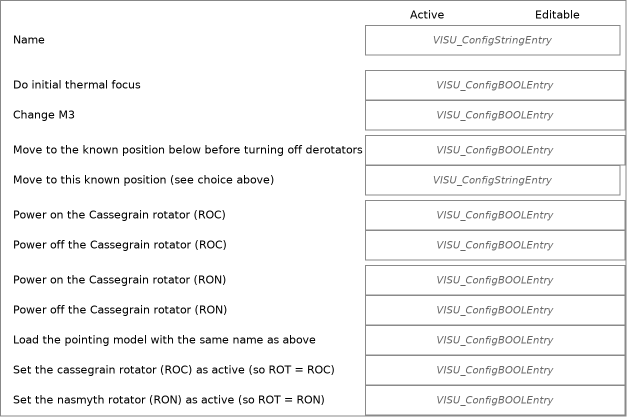
VISUALIZATION VISU_MTCSConfig_Instrument  // 627x417
VAR_IN_OUT
    active : InstrumentConfig;
    editable : InstrumentConfig;
END_VAR
    Label (365,5 125x20), "Active"
    Label (495,5 125x20), "Editable"
    Label (10,25 125x30), "Name"
    Frame (365,25 255x30)
        shows VISU_ConfigStringEntry(active := active.name, editable := editable.name)
    Label (10,70 160x30), "Do initial thermal focus"
    Frame (365,70 260x30)
        shows VISU_ConfigBOOLEntry(active := active.doInitialThermalFocus, editable := editable.doInitialThermalFocus)
    Label (10,100 160x30), "Change M3"
    Frame (365,100 260x30)
        shows VISU_ConfigBOOLEntry(active := active.changeM3, editable := editable.changeM3)
    Frame (365,135 260x30)
        shows VISU_ConfigBOOLEntry(active := active.moveKnownPosition, editable := editable.moveKnownPosition)
    Label (10,135 360x30), "Move to the known position below before turning off derotators"
    Frame (365,200 260x30)
        shows VISU_ConfigBOOLEntry(active := active.powerOnRoc, editable := editable.powerOnRoc)
    Label (10,200 280x30), "Power on the Cassegrain rotator (ROC)"
    Frame (365,165 255x30)
        shows VISU_ConfigStringEntry(active := active.moveKnownPositionName, editable := editable.moveKnownPositionName)
    Label (10,165 340x30), "Move to this known position (see choice above)"
    Frame (365,230 260x30)
        shows VISU_ConfigBOOLEntry(active := active.powerOffRoc, editable := editable.powerOffRoc)
    Label (10,230 350x30), "Power off the Cassegrain rotator (ROC)"
    Frame (365,265 260x30)
        shows VISU_ConfigBOOLEntry(active := active.powerOnRon, editable := editable.powerOnRon)
    Label (10,265 280x30), "Power on the Cassegrain rotator (RON)"
    Frame (365,295 260x30)
        shows VISU_ConfigBOOLEntry(active := active.powerOffRon, editable := editable.powerOffRon)
    Label (10,295 350x30), "Power off the Cassegrain rotator (RON)"
    Frame (365,325 260x30)
        shows VISU_ConfigBOOLEntry(active := active.loadPointingModel, editable := editable.loadPointingModel)
    Label (10,325 360x30), "Load the pointing model with the same name as above"
    Label (10,355 360x30), "Set the cassegrain rotator (ROC) as active (so ROT = ROC)"
    Frame (365,355 260x30)
        shows VISU_ConfigBOOLEntry(active := active.rocActive, editable := editable.rocActive)
    Label (10,385 360x30), "Set the nasmyth rotator (RON) as active (so ROT = RON)"
    Frame (365,385 260x30)
        shows VISU_ConfigBOOLEntry(active := active.ronActive, editable := editable.ronActive)
END_VISUALIZATION

(* stored: Version 1.1.0.1, ProductVersion 3.1.4019.2
   Visu VISU_MTCSConfig_Instrument: Id {cdeb807c-a30c-4dac-a5e4-a7ea4eb9311f} *)
